TYPE ST_Steuerung_auto_manu_BOOL :
STRUCT
	auto			: BOOL;
	manu			: BOOL;
	manu_Modus		: BOOL;
END_STRUCT
END_TYPE

(* stored: Version 1.1.0.1, ProductVersion 3.1.4024.9
   DUT ST_Steuerung_auto_manu_BOOL: Id {1a406012-a05f-42e7-a1a7-50741c9acbc0} *)
